(* PLC project SafeLOGIC-1, BrAutomation SafeDESIGNER  4.3.2.11 *)
(* stored: companyURL http://www.br-automation.com, creationDateTime Tue Mar 20 14:54:59 2018 *)

PROGRAM Main

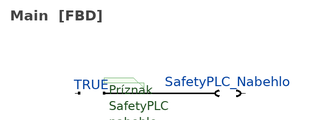
(* FBD diagram, written out as Structured Text *)
(* Príznak SafetyPLC nabehlo *)
SafetyPLC_Nabehlo := TRUE;
END_PROGRAM
